% RSLogix 500 project ANALOG_TANK_PUMP_CONTROL.RSS, saved by version 8.30.00.16 %
PROJECT "UNTITLED"    % processor: Bul.1763 MicroLogix 1100 Series B %

PROGRAM FILES
  LAD 2 "MAIN"  3 rungs
  LAD 3 "IO"  4 rungs  % IO %
  LAD 4 "CONTROL"  6 rungs  % IO %

DATA FILES
  O0 OUTPUT  4 elements
  I1 INPUT  13 elements
  S2 STATUS  66 elements
  B3 BINARY  1 elements
  T4 TIMER  5 elements
  C5 COUNTER  1 elements
  R6 CONTROL  1 elements
  N7 INTEGER  1 elements
  F8 FLOAT  1 elements

LADDER 2 "MAIN"
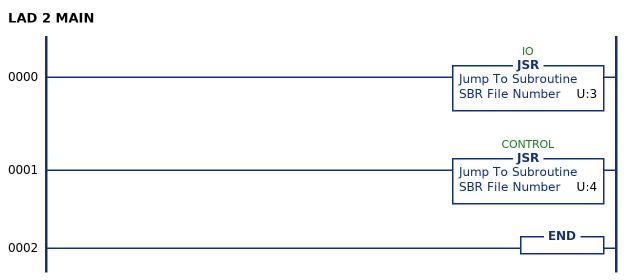
% Rung: 0 %
SOR JSR U:3 EOR
%   U:3  "IO" %
% Rung: 1 %
SOR JSR U:4 EOR
%   U:4  "CONTROL" %
% Rung: 2 %
SOR END EOR

LADDER 3 "IO"    % IO %
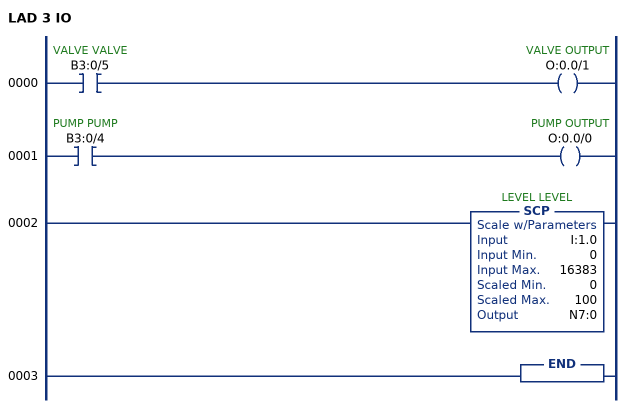
% Rung: 0 %
SOR XIC B3:0/5 OTE O:0.0/1 EOR
%   B3:0/5  VALVE  "VALVE" %
%   O:0.0/1  "VALVE OUTPUT" %
% Rung: 1 %
SOR XIC B3:0/4 OTE O:0.0/0 EOR
%   B3:0/4  PUMP  "PUMP" %
%   O:0.0/0  "PUMP OUTPUT" %
% Rung: 2 %
SOR SCP I:1.0 0 16383 0 100 N7:0 EOR
%   N7:0  LEVEL  "LEVEL" %
% Rung: 3 %
SOR END EOR

LADDER 4 "CONTROL"    % IO %
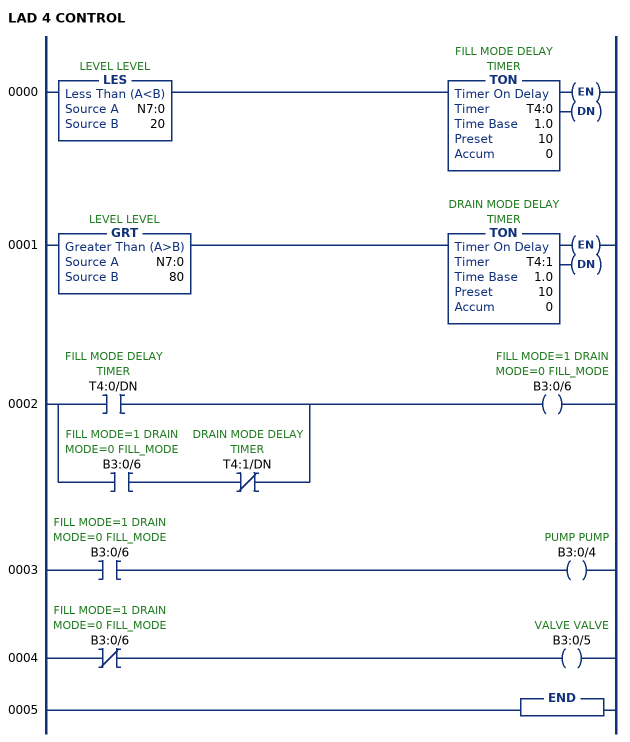
% Rung: 0 %
SOR LES N7:0 20 TON T4:0 1.0 10 0 EOR
%   N7:0  LEVEL  "LEVEL" %
%   T4:0  "FILL MODE DELAY TIMER" %
% Rung: 1 %
SOR GRT N7:0 80 TON T4:1 1.0 10 0 EOR
%   N7:0  LEVEL  "LEVEL" %
%   T4:1  "DRAIN MODE DELAY TIMER" %
% Rung: 2 %
SOR BST XIC T4:0/DN NXB XIC B3:0/6 XIO T4:1/DN BND OTE B3:0/6 EOR
%   T4:0  "FILL MODE DELAY TIMER" %
%   B3:0/6  FILL_MODE  "FILL MODE=1 DRAIN MODE=0" %
%   T4:1  "DRAIN MODE DELAY TIMER" %
% Rung: 3 %
SOR XIC B3:0/6 OTE B3:0/4 EOR
%   B3:0/6  FILL_MODE  "FILL MODE=1 DRAIN MODE=0" %
%   B3:0/4  PUMP  "PUMP" %
% Rung: 4 %
SOR XIO B3:0/6 OTE B3:0/5 EOR
%   B3:0/6  FILL_MODE  "FILL MODE=1 DRAIN MODE=0" %
%   B3:0/5  VALVE  "VALVE" %
% Rung: 5 %
SOR END EOR

OTHER DOCUMENTED ADDRESSES
  B3:0/0  HH_SWITCH  "HH SWITCH"
  B3:0/1  H_SWITCH  "H SWITCH"
  B3:0/2  L_SWITCH  "L SWITCH"
  B3:0/3  LOW_LOW  "LOW LOW"
  I:0.0/0  "HH SWITCH INPUT"
  I:0.0/1  "H SWITCH INPUT"
  I:0.0/2  "L SWITCH INPUT"
  I:0.0/3  "LL SWITCH INPUT"

DATA TABLE (non-zero values as saved)
DATA T4
% .PRE .ACC %
% T4:0 % 10 0
% T4:1 % 10 0
